FUNCTION Matrix_ElementSum : BOOL
VAR_INPUT
	A : REFERENCE TO Matrix;
	B : REFERENCE TO Matrix;
	Res : REFERENCE TO Matrix;
END_VAR
VAR
	I : UINT;
END_VAR

IF NOT(A.IsEqualSize(Res)) OR A.IsEmpty THEN
	Matrix_ElementSum := FALSE;
	RETURN;
END_IF

IF NOT(B.IsEqualSize(Res)) OR B.IsEmpty THEN
	Matrix_ElementSum := FALSE;
	RETURN;
END_IF

Matrix_ElementSum := TRUE;

FOR I := 0 TO Res.Length - 1 DO
	Res.SetI(I,A.GetI(I)+B.GetI(I));
END_FOR

END_FUNCTION

(* stored: Version 1.1.0.1, ProductVersion 3.1.4024.9
   POU Matrix_ElementSum: Id {dd7ad31b-9e72-403d-8fad-fec05d5191bf}, SpecialFunc None *)
